KUKA KRL program: dejar_darsena1.src, dejar_darsena1.dat

--- dejar_darsena1.src ---
&ACCESS RV1
&REL 1316
&COMMENT Dejada Darsena 1
DEF Dejar_Darsena1()

;*************************************************;
;***          DEJAR PRODUCTO EN EL PALE        ***;
;*                                               *;
;*                 Movimientos.                  *;
;*************************************************;




IF  NOT INIT THEN
 ;FOLD INI
 ;FOLD BASISTECH INI
 GLOBAL INTERRUPT DECL 3 WHEN $STOPMESS==TRUE DO IR_STOPM ( )
 INTERRUPT ON 3
 BAS (#INITMOV,0 )
 ;ENDFOLD (BASISTECH INI)
 ;FOLD GRIPPERTECH INI
 ;USER_GRP (0,DUMMY,DUMMY,GDEFAULT )
 ;ENDFOLD (GRIPPERTECH INI)
 ;FOLD USER INI
 ;Make your modifications here

 ;ENDFOLD (USER INI)
   ;ENDFOLD (INI)
   INIT=TRUE
 ENDIF

continue

;CAMBIO DE BASE-->BASE DARSENA 1
  FAPROXIMACION_DEJADA.BASE_NO=2
  FDEJADA.BASE_NO=2
  FSALIDA_DEJADA.BASE_NO=2


;ORI ENTRADA DEJADA==ORI DEJADA
  XENTRADA_DEJADA_DARS1.A=XAPROXIMACION_DEJADA.A
  XENTRADA_DEJADA_DARS1.B=XAPROXIMACION_DEJADA.B
  XENTRADA_DEJADA_DARS1.C=XAPROXIMACION_DEJADA.C
  XENTRADA_DEJADA_DARS1.T=XAPROXIMACION_DEJADA.T

;FOLD PTP ENTRADA_DEJADA_DARS1 CONT Vel=100 % PDAT127 Tool[2]:garras Base[4]:darsena_1;%{PE}%R 5.6.16,%MKUKATPBASIS,%CMOVE,%VPTP,%P 1:PTP, 2:ENTRADA_DEJADA_DARS1, 3:C_PTP, 5:100, 7:PDAT127
$BWDSTART=FALSE
PDAT_ACT=PPDAT1
FDAT_ACT=FENTRADA_DEJADA_DARS1
BAS(#PTP_PARAMS,100)
PTP XENTRADA_DEJADA_DARS1 C_PTP
;ENDFOLD



;FOLD PTP APROXIMACION_DEJADA  Vel=100 % PDAT129 Tool[0] Base[0];%{PE}%R 8.3.22,%MKUKATPBASIS,%CMOVE,%VPTP,%P 1:PTP, 2:aPROXIMACION_DEJADA, 3:, 5:100, 7:PDAT129
$BWDSTART=FALSE
PDAT_ACT=PPDAT1
FDAT_ACT=FAPROXIMACION_DEJADA
BAS(#PTP_PARAMS,100)
PTP xAproximacion_dejada C_PTP
;ENDFOLD

TRIGGER WHEN DISTANCE = 1 DELAY=-100 DO PULSE(ABRIR_GARRAS,TRUE,0.5)

;FOLD LIN DEJADA  Vel=2 m/s CPDAT46 Tool[0] Base[0];%{PE}%R 8.3.22,%MKUKATPBASIS,%CMOVE,%VLIN,%P 1:LIN, 2:DEJADA, 3:, 5:2, 7:CPDAT46
$BWDSTART=FALSE
LDAT_ACT=LCPDAT1
FDAT_ACT=FDEJADA
BAS(#CP_PARAMS,2)
LIN XDEJADA C_DIS
;ENDFOLD

EXTENDER_PISADORES=FALSE

WAIT FOR (GARRAS_ABIERTAS)


TRIGGER WHEN DISTANCE = 1 DELAY=-100 DO PULSE(CERRAR_GARRAS,TRUE,0.1)


;FOLD LIN Salida_DEJADA  Vel=2 m/s CPDAT46 Tool[0] Base[0];%{PE}%R 8.3.22,%MKUKATPBASIS,%CMOVE,%VLIN,%P 1:LIN, 2:DEJADA, 3:, 5:2, 7:CPDAT46
$BWDSTART=FALSE
LDAT_ACT=LCPDAT1
FDAT_ACT=FSalida_DEJADA
BAS(#CP_PARAMS,2)
LIN XSalida_DEJADA C_DIS
;ENDFOLD




;FOLD PTP ENTRADA_DEJADA_DARS1 CONT Vel=100 % PDAT127 Tool[2]:garras Base[4]:darsena_1;%{PE}%R 5.6.16,%MKUKATPBASIS,%CMOVE,%VPTP,%P 1:PTP, 2:ENTRADA_DEJADA_DARS1, 3:C_PTP, 5:100, 7:PDAT127
$BWDSTART=FALSE
PDAT_ACT=PPDAT1
FDAT_ACT=FENTRADA_DEJADA_DARS1
BAS(#PTP_PARAMS,100)
PTP XENTRADA_DEJADA_DARS1 C_PTP
;ENDFOLD



CONTADOR_SACOS_DARSENA1=CONTADOR_SACOS_DARSENA1+1


;FOLD PTP home Vel=100 % PDAT130;%{PE}%R 5.6.16,%MKUKATPBASIS,%CMOVE,%VPTP,%P 1:PTP, 2:home, 3:, 5:100, 7:PDAT130
$BWDSTART=FALSE
PDAT_ACT=PPDAT130
FDAT_ACT=Fhome
BAS(#PTP_PARAMS,100)
$H_POS=XHOME
PTP Xhome
;ENDFOLD
END

--- dejar_darsena1.dat ---
&ACCESS RV1
&REL 1316
&COMMENT Dejada Darsena 1
DEFDAT  DEJAR_DARSENA1 PUBLIC

;FOLD EXTERNAL DECLARATIONS;%{PE}%MKUKATPBASIS,%CEXT,%VCOMMON,%P
;FOLD BASISTECH EXT;%{PE}%MKUKATPBASIS,%CEXT,%VEXT,%P
EXT  BAS (BAS_COMMAND  :IN,REAL  :IN )
DECL INT SUCCESS
;ENDFOLD (BASISTECH EXT)
;FOLD USER EXT;%{E}%MKUKATPUSER,%CEXT,%VEXT,%P
;Make here your modifications

;ENDFOLD (USER EXT)
;ENDFOLD (EXTERNAL DECLARATIONS)




DECL BASIS_SUGG_T LAST_BASIS={POINT1[] "home                    ",POINT2[] "home                    ",CP_PARAMS[] "CPDAT46                 ",PTP_PARAMS[] "PDAT130                 ",CONT[] "                        ",CP_VEL[] "2                       ",PTP_VEL[] "100                     ",SYNC_PARAMS[] "SYNCDAT                 ",SPL_NAME[] "S0                      "}
; DATOS

DECL E6POS XENTRADA_DEJADA_DARS1={X 472.255615,Y 536.637573,Z 1677.927,A 0.0,B 0.0,C -180.0,S 6,T 58,E1 0.0,E2 0.0,E3 0.0,E4 0.0,E5 0.0,E6 0.0}
DECL FDAT FENTRADA_DEJADA_DARS1={TOOL_NO 2,BASE_NO 2,IPO_FRAME #BASE,POINT2[] " ",TQ_STATE FALSE}

DECL PDAT PPDAT1={VEL 100.0,ACC 100.0,APO_DIST 100.0}
DECL LDAT LCPDAT1={VEL 2.0,ACC 100.0,APO_DIST 100.0,APO_FAC 50.0,ORI_TYP #VAR,CIRC_TYP #BASE,JERK_FAC 50.0,EXAX_IGN 0}






DECL PDAT PPDAT130={VEL 100.0,ACC 100.0,APO_DIST 100.0}
ENDDAT
